TYPE ST_OPCUA_NodeVariablePair_BOOL :
STRUCT
	clientVariable : BOOL;
	clientVariableInfo : __SYSTEM.VAR_INFO;
	serverNodeIdentifier : STRING;
END_STRUCT
END_TYPE

(* stored: Version 1.1.0.1, ProductVersion 3.1.4024.9
   DUT ST_OPCUA_NodeVariablePair_BOOL: Id {4aab61c0-be58-40b2-9d49-f114760d457e} *)
